Universal Robots PolyScope program: test1.urp

Program test1 (installation=default directory=/programs/test createdIn=3.14.1.1031110 lastSavedIn=3.14.1.1031110 robotSerialNumber=2018300229)
Calibrated DH parameters: a=[-0.000133, -0.610916, -0.569347, 0.000119, -0.000067, 0]; d=[0.127899, 3.644122, -0.017787, -3.463089, 0.115767, 0.092147]; alpha=[1.570708, -0.011279, -0.012231, 1.568854, -1.569164, 0]; deltaTheta=[-0.000097, -0.067195, -0.010506, 0.077758, -0.000102, -0.000058]
BeforeStart
  s_open := socket_open("192.168.0.10", 30000)
  Loop While (checkContinuously=false) expression=s_open ≟  False
    s_open := socket_open("192.168.0.10", 30000)
Robot Program (runOnlyOnce=false)
  toserver := "robot start"
  Script: socket_send_string(toserver)
  aserver := socket_read_binary_integer(1)
  Wait Sleep waitTime=60
  Popup Message (haltProgram=false message=End inputType=Text)
